// TIA Portal V16 export
// export: Created 2025-08-01T13:38:05.0723434Z, ExportSetting WithDefaults, DisplayName Totally Integrated Automation Portal, DisplayVersion V16, DisplayName TIA Portal Version Control Interface, DisplayVersion V16, DisplayName TIA Portal Openness, DisplayVersion V16, DisplayName STEP 7 Professional, DisplayVersion V16, DisplayName STEP 7 Safety, DisplayVersion V16, DisplayName WinCC Advanced, DisplayVersion V16
DATA_BLOCK "Uitlooptimer_Trilgoten"   // DB11
// stored: AutoNumber true, InstanceOfName TON_SFB, OfSystemLibElement TON, OfSystemLibVersion 1.0
"TON_SFB"
   // VAR_INPUT
   //    IN : Bool;
   //    PT : Time;
   // END_VAR
   // VAR_OUTPUT
   //    Q : Bool;
   //    ET : Time;
   // END_VAR
   // VAR RETAIN
   //    STATE : Byte;
   //    STIME : Time;
   //    ATIME : Time;
   // END_VAR
BEGIN
END_DATA_BLOCK
